// TIA Portal V19 export
DATA_BLOCK "DB_Panel_OVERVIEW"   // DB50
{ S7_Optimized_Access := 'FALSE' }
// stored: AutoNumber false
   VAR
      BA : Struct
         Not_Aus : Bool := FALSE;   // Not-Aus ist betätigt
         free0 : Bool := FALSE;   // sonst Anlage vom PC bedienen, nur bei BA-Schalter auf Auto
         free1 : Bool := FALSE;   // sonst Automatikbetrieb ist nicht freigegeben
         Tippbetrieb : Bool := FALSE;   // Tippbetrieb
         Handbetrieb : Bool := TRUE;   // Handbetrieb
         Automat_ein : Bool := FALSE;   // Automatikbetrieb möglich
         Automat_aus : Bool := FALSE;   // Automatikbetrieb nicht möglich
         Anlauf_Auto : Bool := FALSE;   // Anlauf Automatik für Scanvorgang WT-Positionen auf letzte Automatikposition
         Einfahr_Stop : Bool := FALSE;   // Stoppt die Einfahrt von WT in die Anlage(Feierabendprogramm)
         Mess_on : Bool := FALSE;   // Einmessung aktiv
         Taktwechsel : Bool := FALSE;   // Taktwechsel durchführen
         SIM_HISPEED : Bool := FALSE;   // Simulation erfolgt mit doppelter Geschwindigkeit
         Simulation : Bool := TRUE;   // Simulation eingeschaltet
         COM_RST : Bool := TRUE;   // Complete Restart
         FP_Automat_ein : Bool := FALSE;   // Flankenmerker positive Flanke Taste Automat ein
         newConfig : Bool := FALSE;   // neue Konfiguration (Daten neu verteilen)
      END_STRUCT;
      Offset : Int := 50;
      Leng : Int := 40;
      resW : Word := 16#0000;
      resDW2 : DWord := 16#0000_0000;
      resDW3 : DWord := 16#0000_0000;
      last_Takt : DInt := 0;
      Taktzeit : DInt := 0;   // Zeit die der Takt läuft
      Takt_Ware : DInt := 0;   // Zeit seit Ausfahrt letzte Fertigware
      resW1 : Word := 16#0000;
      Stop_Anlage : Byte := 16#00;   // ungleich 0-->Kettenbearbeitung anhalten
      Feierabend : Byte := 16#00;   // ungleich 0-->FEIERABENDPROGRAMM
      Sonder_BA : Byte := 16#00;   // ungleich 0-->ELEKTROLYSE, ENTMETALLISIEREN
      IST_Sonder_BA : Byte := 16#00;
      FB_FW_akt : Word := 16#0000;   // an Fernbedienung gewählter FW
      SPS_getaktet : Bool := TRUE;
      resDW9 : Word := 16#0000;
      Systime : DInt := 0;
      WT_Frueh : Byte := 16#00;   // Anzeige Anzahl der fertiggestellten WTs in der Frühschicht
      WT_Spaet : Byte := 16#15;   // Anzeige Anzahl der fertiggestellten WTs in der Spätschicht
      WT_Nacht : Byte := 16#00;   // Anzeige Anzahl der fertiggestellten WTs in der Nachtschicht
      resB : Byte := 16#00;
      resI : Int := 0;
      Pos : Array[1..30] of Struct   // * Feldlänge anpassen
         WT_Nr_lang : DInt;   // Warenträger-Nr lang
         WT_Nr_kurz : Byte;   // Warenträger-Nr kurz DB
         Stange_Nr : Byte;   // Warenstangen-Nr. (falls vorhanden)
         Soll_Expo : DInt;   // Sollwert Expositionszeit
         Rest_Expo : DInt;   // Verbleibende Expositionszeit
         BE_rdy : Bool;   // Beladestand bereit
         BE_leer : Bool;   // Beladestand leer
         BE_WT_vorhanden : Bool;   // Beladestand mit nicht aufgebbaren WT belegt
         BE_verriegelt : Bool;   // Beladestand angedockt und verriegelt(arretiert)
         BE_gelb : Bool;
         BE_rot : Bool;
         BE_Charge_ok : Bool;   // Behandlung fehlerfrei
         BE_Charge_nok : Bool;   // Fehler bei Behandlung
         Sonderfkt : Byte;   // Sonderfunktionen frei verwendbar(WT-Kennung)
         priorisiert : Bool;   // priorisierter WT im Bad
         in_Anlage : Bool;   // will in die Anlage
         in_Entm : Bool;   // will in die Entmetallisierung
         aus_Anlage : Bool;   // kommt aus der Anlage
         aus_Entm : Bool;   // kommt aus der Entmetallisierung
         Speicher : Bool;   // Speicherprogramm
         Warnung : Bool;   // in Position wurde eine Warnung ausgelöst
         Alarm : Bool;   // in position wurde ein Alarm ausgelöst
         belegt : Bool;   // Bad belegt
         Trommel : Bool;   // Trommelware im Bad
         Leer_WT : Bool;   // Leerstange im Bad
         Vorruf : Bool;   // Vorruf für Fahrwagen ausgelößt
         fertig : Bool;   // Expozeit abgelaufen WT zu Abholung bereit
         Sperre_in : Bool;   // Einfahrsperre
         Sperre_FW : Bool;   // Überfahrsperre
         Sperre_out : Bool;   // Ausfahrsperre
         Befx : Int;   // Befehlsindex
         Vorsperre : Bool;   // Einfahrsperre angemeldet
         Dummy1 : Bool;   // Dummy auf Dummyposition abgelegt
         Dummy2 : Bool;   // Dummy auf Mittenposition abgelegt
         Dkl_auf_Pos : Bool;   // Deckel auf dieser Position
         Expo_Warn : Bool;   // Warnung: Toleranzüberschreitg.Expozeit
         Expo_Off : Bool;   // Expositionszeit eingefroren
         NSP_ON : Bool;   // Laufanzeige Nachspeisung
         SPR_ON : Bool;   // Laufanzeige Spritzregister
         WT_Typ : Byte;   // Art des Warenträgers (z.Bsp. bei fester Zuordnung Ware-WT)
         Verweilzeit : DInt;   // Verweilzeit in s
         Sonderwert_1 : Real;   // z.B. Gewicht bei Beladestand
         Fertigzeitpunkt : DInt;   // Systemzeit PC, wann WT voraussichtlich fertig
         Sonderwert_2 : Real;   // z.B. Gewicht bei Beladestand
         resb : Byte;
         Dkl_zu : Bool;   // Deckel ist zu
         Dkl_auf : Bool;   // Deckel ist auf
         res392 : Bool;
         res393 : Bool;
         PendelHub : Bool;   // Mehrfachtauchen
         res395 : Bool;
         res396 : Bool;
         res397 : Bool;
      END_STRUCT;
   END_VAR
BEGIN
   Pos[1..30].WT_Nr_lang := 0;
   Pos[1..30].WT_Nr_kurz := 16#00;
   Pos[1..30].Stange_Nr := 16#00;
   Pos[1].Soll_Expo := 0;
   Pos[2].Soll_Expo := 360;
   Pos[3].Soll_Expo := 60;
   Pos[4..7].Soll_Expo := 1260;
   Pos[8..9].Soll_Expo := 90;
   Pos[10].Soll_Expo := 75;
   Pos[11..12].Soll_Expo := 5;
   Pos[13..14].Soll_Expo := 75;
   Pos[15..16].Soll_Expo := 5;
   Pos[17].Soll_Expo := 75;
   Pos[18].Soll_Expo := 5;
   Pos[19].Soll_Expo := 75;
   Pos[20].Soll_Expo := 5;
   Pos[21].Soll_Expo := 10;
   Pos[22].Soll_Expo := 360;
   Pos[23..27].Soll_Expo := 5;
   Pos[28].Soll_Expo := 0;
   Pos[29..30].Soll_Expo := 5;
   Pos[1..30].Rest_Expo := 0;
   Pos[1].BE_rdy := TRUE;
   Pos[2..30].BE_rdy := FALSE;
   Pos[1..30].BE_leer := FALSE;
   Pos[1..30].BE_WT_vorhanden := FALSE;
   Pos[1].BE_verriegelt := TRUE;
   Pos[2..30].BE_verriegelt := FALSE;
   Pos[1..30].BE_gelb := FALSE;
   Pos[1..30].BE_rot := FALSE;
   Pos[1..30].BE_Charge_ok := FALSE;
   Pos[1..30].BE_Charge_nok := FALSE;
   Pos[1..30].Sonderfkt := 16#00;
   Pos[1..30].priorisiert := FALSE;
   Pos[1..30].in_Anlage := FALSE;
   Pos[1..30].in_Entm := FALSE;
   Pos[1..30].aus_Anlage := FALSE;
   Pos[1..30].aus_Entm := FALSE;
   Pos[1..30].Speicher := FALSE;
   Pos[1..30].Warnung := FALSE;
   Pos[1..30].Alarm := FALSE;
   Pos[1..30].belegt := FALSE;
   Pos[1..30].Trommel := FALSE;
   Pos[1..30].Leer_WT := FALSE;
   Pos[1..30].Vorruf := FALSE;
   Pos[1..30].fertig := FALSE;
   Pos[1..30].Sperre_in := FALSE;
   Pos[1..30].Sperre_FW := FALSE;
   Pos[1..30].Sperre_out := FALSE;
   Pos[1..30].Befx := 0;
   Pos[1..30].Vorsperre := FALSE;
   Pos[1..30].Dummy1 := FALSE;
   Pos[1..30].Dummy2 := FALSE;
   Pos[1..30].Dkl_auf_Pos := FALSE;
   Pos[1..30].Expo_Warn := FALSE;
   Pos[1..30].Expo_Off := FALSE;
   Pos[1..30].NSP_ON := FALSE;
   Pos[1..30].SPR_ON := FALSE;
   Pos[1..30].WT_Typ := 16#00;
   Pos[1..30].Sonderwert_1 := 0.0;
   Pos[1..30].Fertigzeitpunkt := 0;
   Pos[1..30].Sonderwert_2 := 0.0;
   Pos[1..30].resb := 16#00;
   Pos[1..30].Dkl_zu := FALSE;
   Pos[1..30].Dkl_auf := FALSE;
   Pos[1..30].res392 := FALSE;
   Pos[1..30].res393 := FALSE;
   Pos[1..30].PendelHub := FALSE;
   Pos[1..30].res395 := FALSE;
   Pos[1..30].res396 := FALSE;
   Pos[1..30].res397 := FALSE;
END_DATA_BLOCK
